Universal Robots URScript: 00B_05_Che_BoXian.script

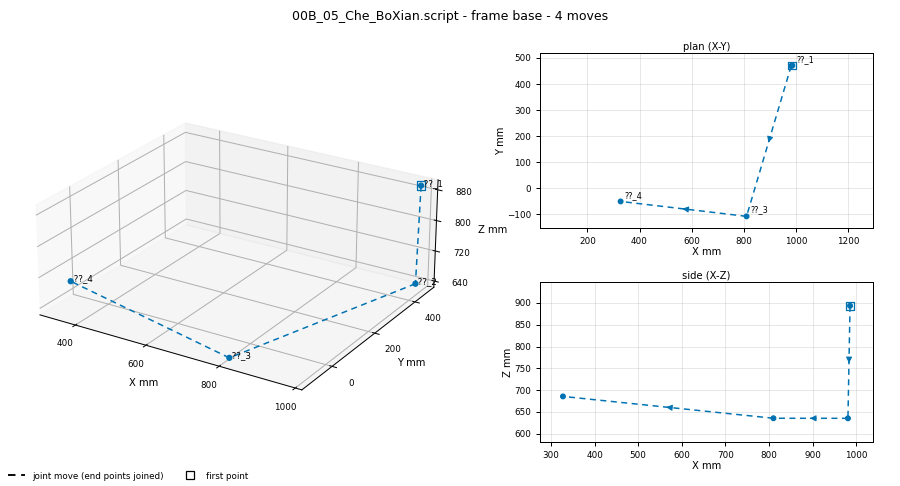
[picture p0: tool path of 00B_05_Che_BoXian.script in frame base, 4 of 4 moves have a stored position in this frame; points joined in program order, loops and branches not executed]
def P00B_05_Che_BoXian():
  set_gravity([0.0, 0.0, 9.82])
  set_safety_mode_transition_hardness(1)
  set_standard_analog_input_domain(0, 1)
  set_standard_analog_input_domain(1, 1)
  set_tool_analog_input_domain(0, 1)
  set_tool_analog_input_domain(1, 1)
  set_analog_outputdomain(0, 0)
  set_analog_outputdomain(1, 0)
  set_tool_voltage(24)
  set_input_actions_to_default()
  set_tcp(p[0.0,0.0,0.32,0.0,0.0,-0.5236])
  set_payload(8.0)
  global Zhua_1=[0.08063, -2.42649, -1.72682, -0.47876, 0.40808, -1.10831]
  global prepose=p[0.98979, -0.16931, -0.39963, 1.98720, 0.07234, 0.05469]
  global i_var_2=0
  global i_var_1=True
  global pose=p[0.98979, -0.31931, -0.39963, 1.98720, 0.07234, 0.05469]
  $ 1 "机器人程序"
  $ 2 "MoveJ"
  $ 3 "路点_1"
  set_tcp(p[0.0,0.0,0.32,0.0,0.0,-0.5236])
  movej(get_inverse_kin(p[.986022577824, .470935745532, .893486716718, .023234474844, .053251665138, 1.539194676148], qnear=[0.5973623394966125, -2.2468321959124964, -1.0992949644671839, -1.4186971823321741, -1.572995964680807, -0.10806590715517217]), a=0.6981317007977318, v=0.5235987755982988)
  $ 4 "路点_2"
  set_tcp(p[0.0,0.0,0.32,0.0,0.0,-0.5236])
  movej(get_inverse_kin(p[.981238934148, .469129670806, .635370749874, .023115886656, .052923633500, 1.536395372295], qnear=[0.5985262989997864, -2.4097216765033167, -1.2966707388507288, -1.0581257979022425, -1.5720375219928187, -0.10803588069844901]), a=0.6981317007977318, v=0.5235987755982988)
  $ 5 "路点_3"
  set_tcp(p[0.0,0.0,0.32,0.0,0.0,-0.5236])
  movej(get_inverse_kin(p[.810237932149, -.107355644838, .635529853043, .034609132840, .041661669177, 1.009701484024], qnear=[0.07159113883972168, -2.0702713171588343, -1.9360860029803675, -0.7575925032245081, -1.5674012343036097, -0.10803588069844901]), a=0.6981317007977318, v=0.5235987755982988)
  $ 6 "路点_4"
  set_tcp(p[0.0,0.0,0.32,0.0,0.0,-0.5236])
  movej(get_inverse_kin(p[.327412679935, -.050152498225, .685634185776, -.037543580370, .083273804954, 1.218388681840], qnear=[0.2738511562347412, -1.1728676001178187, -2.769737784062521, -0.8336046377765101, -1.633601490651266, -0.10535556474794561]), a=0.6981317007977318, v=0.5235987755982988)
end
